Yaskawa INFORM job: S1_90.JBI

/JOB
//NAME S1_90
//POS
///NPOS 0,0,0,0,0,1
///TOOL 0
///POSTYPE ANGLE
///ANGLE
EX00001=90.0000
//INST
///DATE 2025/06/26 07:14
///ATTR SC,RW
///GROUP1 ST1
NOP
MOVJ EX001 VJ=100.00
END
